FUNCTION SubstractMat3 : ARRAY[0..2, 0..2] OF LREAL
VAR_INPUT
	mat1: ARRAY[0..2, 0..2] OF LREAL;
	mat2: ARRAY[0..2, 0..2] OF LREAL;
END_VAR

VAR
	i, j: INT; 
END_VAR

FOR i := 0 TO 2 DO
	FOR j := 0 TO 2 DO
		SubstractMat3[i,j] := mat1[i,j] - mat2[i,j];
	END_FOR
END_FOR

END_FUNCTION

(* stored: Version 1.1.0.1, ProductVersion 3.1.4024.11
   POU SubstractMat3: Id {cda76593-cb69-4fee-98bd-4974fa426267}, SpecialFunc None *)
